PROGRAM MAIN
VAR
END_VAR

END_PROGRAM

(* stored: Version 1.1.0.1, ProductVersion 3.1.4024.9
   POU MAIN: Id {01b9e83c-3c93-0a70-347c-5bc9962393e7}, SpecialFunc None *)
